// TIA Portal V19 export
VAR_GLOBAL   // PLC tag table "Default tag table"
   Fill_tank AT %M0.0 : Bool;
   Empty_tank AT %M0.1 : Bool;
   BottomDrySensor AT %I0.2 : Bool;
   TopDrySensor AT %I0.3 : Bool;
   BottomValveOpen AT %I0.4 : Bool;
   BottomValveClosed AT %I0.5 : Bool;
   TopValveOpen AT %I0.6 : Bool;
   TopValveClosed AT %I0.7 : Bool;
END_VAR
